Staubli VAL3: PLC.pjx

--- PLC.pjx ---
Parameters version=s7.8 stackSize=5000 millimeterUnit=true
Program file=Main.pgx
Program file=_HomeWatchDog.pgx
Program file=_resetProgram.pgx
Program file=cycle_clearList.pgx
Program file=cycle_end.pgx
Program file=cycle_getList.pgx
Program file=cycle_getLoop.pgx
Program file=cycle_getProg.pgx
Program file=cycle_getSize.pgx
Program file=cycle_isFound.pgx
Program file=cycle_isLock.pgx
Program file=cycle_isPause.pgx
Program file=cycle_isRun.pgx
Program file=cycle_lock.pgx
Program file=cycle_pause.pgx
Program file=cycle_putProg.pgx
Program file=cycle_resume.pgx
Program file=cycle_searchPrg.pgx
Program file=cycle_setLoop.pgx
Program file=cycle_start.pgx
Program file=cycle_stop.pgx
Program file=cycle_unLock.pgx
Program file=cycle_updateLst.pgx
Program file=getJointData.pgx
Program file=getPointData.pgx
Program file=goHome.pgx
Program file=isHome.pgx
Program file=kill.pgx
Program file=pallet_getList.pgx
Program file=pallet_getPos.pgx
Program file=pallet_reset.pgx
Program file=pallet_resetAll.pgx
Program file=pallet_setPos.pgx
Program file=receive.pgx
Program file=send.pgx
Program file=session_change.pgx
Program file=session_get.pgx
Program file=session_search.pgx
Data file=PLC.dtx
Library alias=cycleStatus path=Disk://cycleStatus/cycleStatus.pjx autoload=true password=
Library alias=saveData path=Disk://saveData/saveData.pjx autoload=true password=
Library alias=processList path=Disk://kernel/processList/processList.pjx autoload=true password=
Library alias=OnEvent path=Disk://OnEvent/OnEvent.pjx autoload=true password=
Library alias=use path=Disk://kernel/userPage/userPage.pjx autoload=true password=
Library alias=jt path=Disk://kernel/template/session/saveTraj/JPOINT/JPOINT.pjx autoload=true password=
Library alias=prog path=Disk://instruction/PROG/PROG.pjx autoload=true password=
Library alias=pallet path=Disk://trajectory/PALLET/PALLET.pjx autoload=true password=
Library alias=pt path=Disk://kernel/template/session/saveTraj/POINT/POINT.pjx autoload=true password=
Library alias=tt path=Disk://kernel/template/session/saveTraj/TRAJ/TRAJ.pjx autoload=true password=
Library alias=language path=Disk://kernel/language/language.pjx autoload=true password=
Library alias=gohome path=Disk://goHome/goHome.pjx autoload=true password=
Type name=TrajJoint path=Disk://kernel/template/TrajJoint/TrajJoint.pjx
Type name=TrajectoryItem path=Disk://kernel/template/TrajectoryItem/TrajectoryItem.pjx
Type name=TrajPointItem path=Disk://kernel/template/TrajPointItem/TrajPointItem.pjx
Type name=TrajItem path=Disk://kernel/template/TrajItem/TrajItem.pjx
Type name=FrameItem path=Disk://kernel/template/FrameItem/FrameItem.pjx

--- PLC.dtx ---
public num nToSuperV
string sProgList
string sPresetList
string listProgram
public jointRx jHome
public mdesc nom_speed = {rmax=9999, blend=off}
string sSessionList
string sPalletName
string sSession
string sSession2
dio dOutRobIsReady = {link=ApplicomIO-1\TOPIC1_A-BLOCKA\%Q1}
dio dOutRobInHome = {link=ApplicomIO-1\TOPIC1_A-BLOCKA\%Q0}
dio dOutRobCycle = {link=ApplicomIO-1\TOPIC1_A-BLOCKA\%Q2}
dio dOutRobErr = {link=ApplicomIO-1\TOPIC1_A-BLOCKA\%Q4}
dio dInCycle = {link=ApplicomIO-1\TOPIC1_A-BLOCKA\%I0}
bool bError
aio aSelect = {link=ApplicomIO-1\TOPIC1_A-BLOCKA\%IW8}
num nProgCode
string sProgName
dio dInPlcErr = {link=ApplicomIO-1\TOPIC1_A-BLOCKA\%I1}
dio dOutGunOn = {link=valve1}
dio dOutJobDone
dio dInGohome = {link=ApplicomIO-1\TOPIC1_A-BLOCKA\%I4}
dio dInPauseCycle = {link=ApplicomIO-1\TOPIC1_A-BLOCKA\%I2}
dio dInResumeCycle = {link=ApplicomIO-1\TOPIC1_A-BLOCKA\%I3}
dio dIndisablepower = {link=ApplicomIO-1\TOPIC1_A-BLOCKA\%I5}
dio dOutPauseCycle = {link=ApplicomIO-1\TOPIC1_A-BLOCKA\%Q3}
public aio aTime = {link=ApplicomIO-1\TOPIC1_A-BLOCKA\%QW8}
public aio aSudu = {link=ApplicomIO-1\TOPIC1_A-BLOCKA\%IW10}

--- Main.pgx ---
public program Main()
begin
  wait(nToSuperV==-1)
  // wait the session has been loaded
  watch(saveData:bToReload==true,10)
  watch(saveData:bToReload==false,10)
  //
  logMsg("[KERNEL] PLC:LOAD")
  // Init
  // Clean the process List
  //  call cycle_clearList(0)
  //  call cycle_clearList(1)
  //  call cycle_clearList(2)
  // Reset the loop
  // call cycle_setLoop(false)
  // reload the program LIST
  call cycle_updateLst()
  // set the PLC enable in order to wait a new program in the process LIST without END it
  saveData:bPlcEnable=false
  // get the list of session
  call saveData:getListSession(sSessionList)
  // HOME PARAMETER
  // radius home to check for the best J4-J5-J6 config
  saveData:nRadiusHome=400
  // Set to use or not the HOME position before START the production
  saveData:bNoUseHome=false
  // set to search inside the joints with the same actual config or not
  saveData:bUseHomeConfig=false
  // set to scan the best point along the home trajectory or to attach only to a joint point
  saveData:bUseHomeScanner=true
  while true
    //
    //  SEND TO PLC
    //
    call send()
    //
    //  RECEIVE FROM PLC
    //
    call receive()
    //
    delay(0)
  endWhile
end

--- _HomeWatchDog.pgx ---
public program _HomeWatchDog()
begin
  if taskStatus("resetProgram")!=-1
    //过滤硬件波动
    //    if watch(cycleStatus:bIsHome==true,0)
    if watch(dInGohome==true,0)
    else
      stopMove()
      taskKill("resetProgram")
      watch(taskStatus("resetProgram")==-1,1)
      resetMotion()
    endIf
    if taskStatus("resetProgram")>1
      if taskStatus("resetProgram")>=150 and taskStatus("resetProgram")<=154
        popUpMsg("运动无法到达，超限")
      else
        logMsg("[KERNEL] SUPERVISOR:Task resetProgram problem")
        call OnEvent:OnCycleEvent(12)
      endIf
      stopMove()
      taskKill("resetProgram")
      watch(taskStatus("resetProgram")==-1,1)
      resetMotion()
    endIf
  endIf
end

--- _resetProgram.pgx ---
public program _resetProgram()
begin
  if !cycleStatus:bCycle and !cycleStatus:bPause
    if !cycleStatus:bIsHome
      if taskStatus("resetProgram")==-1
          taskCreate "resetProgram",99,gohome:GOHOME()
     //   watch(taskStatus("resetProgram")==1,1)
        wait(taskStatus("resetProgram")==1)
      endIf
    endIf
  endIf
end

--- cycle_clearList.pgx ---
program cycle_clearList(num x_nType (dimensions=1))
begin
  logMsg("[KERNEL] PLC:Clear list")
  //
  call processList:deleteAll(x_nType)
end

--- cycle_end.pgx ---
program cycle_end()
begin
  if !cycleStatus:bToEnd and cycleStatus:bCycle
    logMsg("[KERNEL] PLC:End cycle")
    call OnEvent:endCycle()
  endIf
end

--- cycle_getList.pgx ---
program cycle_getList(num x_nType (dimensions=1))
  local num i
  local num nSize
  local string sName
begin
  //
  // Get the Cycle process list and put in the
  // global variable listProgram
  //
  // build the list
  nSize=size(listProgram)
  for i=1 to nSize-1
    delete(listProgram[0])
  endFor
  call cycle_getSize(nSize,x_nType)
  call cycle_getProg(sName,1,x_nType)
  // copy the list
  listProgram=sName
  if nSize>0
    for i=1 to nSize-1
      call cycle_getProg(sName,i+1,x_nType)
      insert(listProgram[i])
      listProgram[i]=sName
    endFor
  endIf
  //
end

--- cycle_getLoop.pgx ---
program cycle_getLoop(bool& x_bLoop[] (dimensions=1))
begin
  // get the loop
  call processList:getLoop(x_bLoop)
end

--- cycle_getProg.pgx ---
program cycle_getProg(string& x_sName[] (dimensions=1), num x_nIndex (dimensions=1), num x_nType (dimensions=1))
  local num l_nID
  local num l_nSize[3]
begin
  //
  // get the programm name of the specific
  // x_nIndex, return "" if there is an error
  // x_nIndex start from 1 o N
  //
  if saveData:bDebug
    ? "[KERNEL] PLC:Ask program name at index:"+toString("",x_nIndex)
  endIf
  call cycle_getSize(l_nSize,x_nType)
  if x_nIndex<=l_nSize and x_nIndex>0
    l_nID=0
    call processList:getCycle(x_sName,l_nID,l_nID,x_nIndex-1,x_nType)
  else
    logMsg("[KERNEL] PLC: "+x_sName+" error on the index "+toString("",x_nIndex))
    x_sName=""
  endIf
end

--- cycle_getSize.pgx ---
program cycle_getSize(num& x_nSize[] (dimensions=1), num x_nType (dimensions=1))
  local num l_nID
  local string sName
begin
  //
  // get the size of process list running
  //
  l_nID=0
  call processList:getCycle(sName,l_nID,l_nID,0,x_nType)
  // check if the name is not null
  if sName!=""
    call processList:getSize(x_nSize,x_nType)
  else
    x_nSize=0
  endIf
end

--- cycle_isFound.pgx ---
program cycle_isFound(string x_sProgName (dimensions=1), bool& x_bFound[] (dimensions=1))
  local num i
begin
  x_bFound=false
  // verify if a program is in the program list
  // libList(saveData:sPathProg[0],sProgList)
  // check inside the program List
  for i=0 to size(sProgList)-1
    if sProgList[min(size(sProgList)-1,i)]==x_sProgName
      x_bFound=true
      return
    endIf
  endFor
end

--- cycle_isLock.pgx ---
program cycle_isLock(bool& x_bLock[] (dimensions=1))
begin
  //
  // ask for the PLC lock status
  //
  x_bLock=cycleStatus:bPausePLC
end

--- cycle_isPause.pgx ---
program cycle_isPause(bool& x_bPause[] (dimensions=1))
begin
  //
  // ask for pause status
  //
  x_bPause=cycleStatus:bPause
end

--- cycle_isRun.pgx ---
program cycle_isRun(bool& x_bStatus[] (dimensions=1))
begin
  //
  // ask for the cycle running
  //
  x_bStatus=cycleStatus:bCycle
end

--- cycle_lock.pgx ---
program cycle_lock()
begin
  //
  // Lock by PLC THE CYCLE
  //
  if !cycleStatus:bPausePLC
    logMsg("[KERNEL] PLC:Lock the cycle")
    // lock it
    cycleStatus:bPausePLC=true
    stopMove()
    call OnEvent:OnCycleEvent(2)
    //
  endIf
  //
end

--- cycle_pause.pgx ---
program cycle_pause()
begin
  //
  // PAUSE THE CYCLE
  //
  if !cycleStatus:bPause
    logMsg("[KERNEL] PLC:pause cycle")
    // pause
    cycleStatus:bToPause=true
    watch(cycleStatus:bToPause==false,1)
    //
  endIf
  //
end

--- cycle_putProg.pgx ---
program cycle_putProg(string x_sName (dimensions=1), num x_nType (dimensions=1))
  local bool l_bFound
begin
  //
  // insert one program at the end of the process List
  // 0 -start list
  // 1 -production list
  // 2 -end list
  //
  if saveData:bDebug
    logMsg("[KERNEL] PLC:Insert program: "+x_sName)
  endIf
  // check before if exist
  call cycle_isFound(x_sName,l_bFound)
  if l_bFound
    call processList:insertCycle(-1,x_sName,1,0,x_nType)
    // check to save or not in order to have the same process next boot
    // call processList:save()
  elseIf saveData:bDebug
    ? "[KERNEL] PLC: "+x_sName+" not found in the program List"
  endIf
end

--- cycle_resume.pgx ---
program cycle_resume()
begin
  // resume from PAUSE
  if cycleStatus:bPause==true
    //raise the bit
    cycleStatus:bToPause=true
    watch(cycleStatus:bToPause==false,1)
    // OnEvent
    call OnEvent:OnCycleEvent(3)
  endIf
end

--- cycle_searchPrg.pgx ---
program cycle_searchPrg(num x_nProg (dimensions=1), string& x_sProgName[] (dimensions=1), bool& x_bFound[] (dimensions=1))
  local num i
  local bool l_bOk
  local num l_nChar
  local num l_nProg
begin
  // init
  x_bFound=false
  x_sProgName=""
  //
  // get the list
  //
  // libList(saveData:sPathProg[0],sProgList)
  //
  // search the program from a number:
  //
  // "number+space+name"
  //
  // 01 MyPart
  // 10 YourPart
  //
  for i=0 to size(sProgList)-1
    if sProgList[i]!=""
      toNum(sProgList[i],l_nProg,l_bOk)
      if l_bOk and l_nProg==x_nProg
        x_sProgName=sProgList[i]
        x_bFound=true
        i=size(sProgList)-1
      endIf
    endIf
  endFor
end

--- cycle_setLoop.pgx ---
program cycle_setLoop(bool x_bLoop (dimensions=1))
begin
  logMsg("[KERNEL] PLC:Change loop status")
  call processList:setLoop(x_bLoop)
end

--- cycle_start.pgx ---
program cycle_start()
  local num l_nID
  local num l_nId
  local string l_sName
begin
  //
  // Start the cycle
  //
  call processList:getCycle(l_sName,l_nID,l_nID,0,1)
  if l_sName!=""
    logMsg("[KERNEL] PLC:Start Cycle")
    nToSuperV=0
    wait(nToSuperV==-1)
  endIf
end

--- cycle_stop.pgx ---
program cycle_stop()
begin
  logMsg("[KERNEL] PLC:Stop Cycle")
  if cycleStatus:bCycle or cycleStatus:bSimulation
    // stop bit
    cycleStatus:bToStop=true
    watch(cycleStatus:bToStop==false,1)
  endIf
end

--- cycle_unLock.pgx ---
program cycle_unLock()
begin
  // resume from the Lock
  if cycleStatus:bPausePLC==true
    cycleStatus:bPausePLC=false
    // OnEvent
    call OnEvent:OnCycleEvent(3)
  endIf
end

--- cycle_updateLst.pgx ---
program cycle_updateLst()
  local num i
  local num l_nSize
  local string l_sEvent
begin
  // get the list
  //
  call prog:getSize(l_nSize)
  resize(sProgList,1,l_nSize)
  sProgList=""
  for i=0 to l_nSize-1
    call prog:get(l_sEvent,i)
    // patch for the #program
    sProgList[i]=l_sEvent
  endFor
end

--- getJointData.pgx ---
public program getJointData(string x_sItem (dimensions=1), num x_nIndex (dimensions=1), joint& x_jJoint (dimensions=1), bool& x_bResult (dimensions=1))
  local num i
  local num l_nResult
  local string l_sSession
begin
  // get the joint data from the specific session...
  x_bResult=false
  call saveData:getSession(l_sSession)
  // get the colletion type...
  if sSession!=l_sSession
    // copy back
    sSession=l_sSession
    // load the actual one
    l_nResult=jt:libLoad(saveData:sPathTraj+"JPOINT")
    delay(0)
  endIf
  // use the type...
  if l_nResult==0 and isDefined(jt:tTraj[x_sItem]) and size(jt:tTraj[x_sItem].tData.jJoint)>x_nIndex
    // get the JOINT DATA
    x_jJoint=jt:tTraj[x_sItem].tData.jJoint[x_nIndex]
    delay(0)
    x_bResult=true
  endIf
end

--- getPointData.pgx ---
public program getPointData(string x_sItem (dimensions=1), num x_nIndex (dimensions=1), point& x_pPoint (dimensions=1), bool& x_bResult (dimensions=1))
  local num i
  local num l_nResult
  local string l_sSession
begin
  // get the joint data from the specific session...
  x_bResult=false
  call saveData:getSession(l_sSession)
  // get the colletion type...
  if sSession2!=l_sSession
    // copy back
    sSession2=l_sSession
    // load the actual one
    l_nResult=pt:libLoad(saveData:sPathTraj+"POINT")
    delay(0)
  endIf
  // use the type...
  if l_nResult==0 and isDefined(pt:tTraj[x_sItem]) and size(pt:tTraj[x_sItem].tData.pPoint)>x_nIndex
    // get the JOINT DATA
    x_pPoint=pt:tTraj[x_sItem].tData.pPoint[x_nIndex]
    delay(0)
    x_bResult=true
  endIf
end

--- goHome.pgx ---
program goHome()
begin
  // go to HOME
  // check if the robot is not in cycle
  if !(cycleStatus:bCycle or cycleStatus:bSimulation)
    cycleStatus:bToHome=true
    watch(cycleStatus:bToHome==false,3)
    // wait end of HOME
    watch(cycleStatus:bIsHome,3)
    waitEndMove()
    watch(cycleStatus:bSimulation==false,3)
  endIf
end

--- isHome.pgx ---
program isHome(bool& x_bHome[] (dimensions=1))
begin
  //
  // ask for home status
  //
  x_bHome=cycleStatus:bIsHome
end

--- kill.pgx ---
public program kill()
begin
  // kill the task create in task PLC and reset the signal
  saveData:bPlcEnable=false
end

--- pallet_getList.pgx ---
program pallet_getList()
  local num i
  local num l_nSize
  local string l_sItem
begin
  // get the full pallet list, copy into sPalletName
  call pallet:getSize(l_nSize)
  if size(sPalletName)!=l_nSize
    resize(sPalletName,1,l_nSize)
  endIf
  for i=0 to l_nSize-1
    call pallet:get(l_sItem,i)
    sPalletName[i]=l_sItem
  endFor
end

--- pallet_getPos.pgx ---
program pallet_getPos(string x_sPalletName (dimensions=1), num& x_nPos (dimensions=1))
begin
  // get the actual position of the x_sPalletName
  call pallet:getPalletPos(x_sPalletName,x_nPos)
end

--- pallet_reset.pgx ---
program pallet_reset(string x_sPalletName (dimensions=1))
begin
  // reset the index of the x_sPalletName
  call pallet:setPalletPos(x_sPalletName,0)
end

--- pallet_resetAll.pgx ---
program pallet_resetAll()
begin
  // resetAll the pallet
  call pallet_resetAll()
end

--- pallet_setPos.pgx ---
program pallet_setPos(string x_sPalletName (dimensions=1), num x_nPos (dimensions=1))
begin
  // set the position of the x_sPalletName to x_nPos
  call pallet:setPalletPos(x_sPalletName,x_nPos)
end

--- receive.pgx ---
program receive()
  local num l_nProg
  local string l_sProgName
  local num i
  local bool l_bResult
  local bool l_bRun
  local num l_nSize
  local bool l_bLoaded
  local bool l_bFound
  local string l_sMessage
begin
  //输入参考
  //正常生产
  if dInCycle==true and bError==false
    if esStatus()!=2 and !cycleStatus:bSimulation and cycleStatus:bIsHome and !cycleStatus:bCycle  and workingMode()==4
      nProgCode=aioGet(aSelect)
      call cycle_updateLst()
      call cycle_searchPrg(nProgCode,sProgName,l_bFound)
      if l_bFound
        call cycle_clearList(1)
        call cycle_putProg(sProgName,1)
        call cycle_start()
        logMsg("开始程序-"+sProgName)
        delay(1)
      else
        // no program in the process List
        if workingMode()==1
          call language:message(l_sMessage,91)
          popUpMsg(l_sMessage)
        endIf
      endIf
    endIf
  endIf


  //Pause
  if cycleStatus:bCycle and !cycleStatus:bPause
    if dInPauseCycle==true
      logMsg("暂停程序-"+sProgName)
      call OnEvent:pauseCycle()
    endIf
    //RESUME
  elseIf cycleStatus:bCycle and cycleStatus:bPause
    if dInResumeCycle==true
      logMsg("重启程序-"+sProgName)
      call OnEvent:resumeCycle()
    endIf
  endIf

  if dIndisablepower==true
    if workingMode()==4
      disablePower()
    endIf
    endIf

  //停止生产
  if dInPlcErr==true
    bError=true
    if cycleStatus:bCycle
      logMsg("停止程序-"+sProgName)
      call OnEvent:stopCycle()
      cycleStatus:bToStop=true
      call OnEvent:OnCycleEvent(5)
      call language:message(l_sMessage,-84)
      call use:timerDialog(l_sMessage,1)
      watch(cycleStatus:bToStop==false,1)
    if workingMode()==4
      disablePower()
    endIf
      //      dOutGunOn=false
      //      dOutJobDone=false
    endIf
  else
    bError=false
  endIf

  if dInGohome==true
    if cycleStatus:bIsHome==true
      dOutGunOn=false
      popUpMsg("123")
    endIf
    if !isPowered()
      cycleStatus:bAutoON=true
    endIf
    if watch(isPowered()==true,2)
      call _resetProgram()
    endIf
  else
    call _HomeWatchDog()
  endIf

  if getMonitorSpeed()>=0 and getMonitorSpeed()<101
  if getMonitorSpeed()!=aioGet(aSudu)
    setProfile("Robot","")
    setMonitorSpeed(aioGet(aSudu))
    waitEndMove()
    setProfile("maintenance","spec_cal")
  endIf
  endIf
end

--- send.pgx ---
program send()
begin
  if 4==workingMode() and esStatus()!=2 and cycleStatus:bIsHome and !cycleStatus:bCycle
    dOutRobIsReady=true
  else
    dOutRobIsReady=false
  endIf
  //检查机器是否在home位置
  if cycleStatus:bIsHome
    dOutRobInHome=true
  else
    dOutRobInHome=false
  endIf
  //检查机器人是否有生产程序在执行
  if cycleStatus:bCycle
    dOutRobCycle=true
  else
    dOutRobCycle=false
  endIf

  //急停触发
  if esStatus()==2
    dOutRobErr=true
  else
    dOutRobErr=false
  endIf

//机器人是否处于暂停状态
  if cycleStatus:bPause==true
		dOutPauseCycle=true
	else
    dOutPauseCycle=false
  endIf
  aioSet(aTime,cycleStatus:nCycleTime)
end

--- session_change.pgx ---
program session_change(string x_sName (dimensions=1), bool& x_bResult (dimensions=1))
  local num i
  local string l_sEmpty
  local string l_sEvent
begin
  // check if exist
  // clean the string
  l_sEmpty=""
  x_bResult=false
  if cycleStatus:bCycle==false and cycleStatus:bSimulation==false
    // search inside the sSession
    for i=0 to size(sSessionList)-1
      if x_sName==sSessionList[i]
        // the session exist
        call saveData:changeSession(x_sName)
        // reload the processList
        call processList:loadProcessList(i)
        if i!=0
          popUpMsg("error loading: "+toString("",i))
        else
          // the session has been changed
          x_bResult=true
        endIf
        //
        if !x_bResult
          // not found
          popUpMsg("session not FOUND....")
        endIf
        // reset the homing trajectory
        cycleStatus:bHomeLoaded=false
        // refresh
        use:bUseRefresh=true
        return
      endIf
    endFor
  endIf
  //
end

--- session_get.pgx ---
program session_get(string& x_sName (dimensions=1))
  local num i
  local string l_sEmpty
  local string l_sEvent
begin
  //
  // get the actual session...
  //
  call saveData:getSession(x_sName)
  //
end

--- session_search.pgx ---
program session_search(num x_nSession (dimensions=1), string& x_sSessionName[] (dimensions=1), bool& x_bFounded[] (dimensions=1))
  local num i
  local bool l_bOk
  local num l_nChar
  local num l_nSession
  local string l_sEmpty
begin
  // init
  x_bFounded=false
  x_sSessionName=""
  //
  // get the list
  //
  l_sEmpty=""
  call use:stringCopy(l_sEmpty,sSessionList)
  // get the list of session
  call saveData:getListSession(sSessionList)
  //
  // search the program from a number:
  //
  // "number+space+name"
  //
  // 01 MyPart
  // 10 YourPart
  //
  for i=0 to size(sSessionList)-1
    if sSessionList[i]!=""
      // convert the string "00 name" into a num
      toNum(sSessionList[i],l_nSession,l_bOk)
      if l_bOk and l_nSession==x_nSession
        x_sSessionName=sSessionList[i]
        x_bFounded=true
        // exit
        i=size(sSessionList)-1
      endIf
    endIf
  endFor
end
